(* IEC 61131-3 sources: SmartGondolaPLC/Prog/pous/function-blocks, 1 file *)

(* ---- Test.st ---- *)
FUNCTION_BLOCK Test
VAR_INPUT
	Input : bool;
END_VAR

VAR_OUTPUT
	Output : bool;
END_VAR

Output := Input;

END_FUNCTION_BLOCK
